{attribute 'qualified_only' := ''}
{attribute 'strict' := ''}
TYPE MC_SYNC_MODE :
(
	enum_member := 0
);
END_TYPE

(* stored: Version 1.1.0.1, ProductVersion 3.1.4024.12
   DUT MC_SYNC_MODE: Id {7437c518-137b-4a8f-9065-0ed0d228dcb8} *)
